FUNCTION_BLOCK FB_Manipulatormodul
VAR_INPUT
	bEnable : BOOL;
	bExecute : BOOL;
	
	pXhome : REAL;
	pYhome : REAL;
	pZhome : REAL;
	
	pXconv : REAL;
	pYconv : REAL;
	pZconv : REAL;
	
	pXscale : REAL;
	pYscale : REAL;
	pZscale : REAL;
	
	pXheat : REAL;
	pYheat : REAL;
	pZheat : REAL;
	
	pX1stor : REAL;
	pX2stor : REAL;
	pX3stor : REAL;
	pX4stor : REAL;
	pYstor : REAL;
	pZstor : REAL;
	
	estateE : eBetriebszustand;
	
	bxEndschalter: BOOL;
	byEndschalter: BOOL;
	bzEndschalter: BOOL;
	bGEndschalter: BOOL;
	
END_VAR
VAR_OUTPUT
	estate : eBetriebszustand;
END_VAR
VAR
	fbRobotsteuerung : FB_Robotsteuerung;
	fbTON : TON;
	nstate : INT := 0;
	
	targX   : REAL;
  	targY   : REAL;
 	targZ   : REAL;
  	goRobot : BOOL;
END_VAR
VAR_IN_OUT
    // Achsen-Referenzen 
    ax_ManX    : AXIS_REF;   
    ax_ManY    : AXIS_REF;   
    ax_ManZ    : AXIS_REF;  
	ax_ManG    : AXIS_REF;   
END_VAR

fbRobotsteuerung(
	bEnable:= , 
	bExecute:= goRobot, 
	bxposition:= targX, 
	byposition:= targY, 
	bzposition:= targZ, 
	bxEndschalter:= bxEndschalter, 
	byEndschalter:= byEndschalter, 
	bzEndschalter:= bzEndschalter, 
	bGEndschalter:= bGEndschalter, 
	estate=> , 
	movedone=> , 
	ax_ManX:= ax_ManX, 
	ax_ManY:= ax_ManY, 
	ax_ManZ:= ax_ManZ, 
	ax_ManG:= ax_ManG);
	
	fbTON(IN:= , PT:=T#10S , Q=> , ET=> );
CASE nstate OF 
	0: //off
	estate := eBetriebszustand.off;
	fbRobotsteuerung.bEnable := FALSE;
	
	IF bEnable THEN
		nstate := 10;
	END_IF
	
	10: //Init
	estate := eBetriebszustand.init;
	fbRobotsteuerung.bEnable := TRUE;
	
	IF fbRobotsteuerung.estate = eBetriebszustand.ready THEN
		nstate := 20;
	END_IF
	
	20: //Ready
	estate := eBetriebszustand.ready;
	fbRobotsteuerung.bEnable := TRUE;
	
	IF bExecute THEN
		nState := 30; 
	END_IF
	
	30: //Move to Conveyer
	estate := eBetriebszustand.production;
	targX   := pXconv;
  	targY   := pYconv;
 	targZ   := pZconv;
  	goRobot := TRUE;
	
	IF fbRobotsteuerung.estate = eBetriebszustand.done AND
		estateE = eBetriebszustand.done THEN
		goRobot := FALSE;
		nstate := 40;
	END_IF
	
	40: //Lift Z Achse
	estate := eBetriebszustand.production;
	targX   := pXconv;
  	targY   := pYconv;
 	targZ   := pZhome;
  	goRobot := TRUE;


	IF fbRobotsteuerung.estate = eBetriebszustand.done THEN
		goRobot := FALSE;
		nstate := 50;
	END_IF
	
	50: //scale
	estate := eBetriebszustand.production;
	targX   := pXscale;
  	targY   := pYscale;
 	targZ   := pZscale;
  	goRobot := TRUE;
	fbTON.IN := TRUE;

	IF fbRobotsteuerung.estate = eBetriebszustand.done AND
		fbTON.Q = TRUE THEN
		fbTON.IN := FALSE;
		goRobot := FALSE;
		nstate := 60;
	END_IF
	
	60: //Lift Z Achse
	estate := eBetriebszustand.production;
	targX   := pXscale;
  	targY   := pYscale;
 	targZ   := pZhome;
  	goRobot := TRUE;

	IF fbRobotsteuerung.estate = eBetriebszustand.done THEN
		goRobot := FALSE;
		nstate := 70;
	END_IF
	
	70: //heat
	estate := eBetriebszustand.production;
	targX   := pXheat;
  	targY   := pYheat;
 	targZ   := pZheat;
  	goRobot := TRUE;
	fbTON.IN := TRUE;
	
	IF fbRobotsteuerung.estate = eBetriebszustand.done AND
		fbTON.Q = TRUE THEN
		fbTON.IN := FALSE;
		goRobot := FALSE;
		nstate := 80;
	END_IF

	80: //Lift Z Achse
	estate := eBetriebszustand.production;
	targX   := pXheat;
  	targY   := pYheat;
 	targZ   := pZhome;
  	goRobot := TRUE;

	IF fbRobotsteuerung.estate = eBetriebszustand.done THEN
		goRobot := FALSE;
		nstate := 90;
	END_IF
	
	90: //storage
	estate := eBetriebszustand.production;
	targX   := pX1stor;
  	targY   := pYstor;
 	targZ   := pZstor;
  	goRobot := TRUE;
	fbTON.IN := TRUE;

	IF fbRobotsteuerung.estate = eBetriebszustand.done AND
		fbTON.Q = TRUE THEN
		fbTON.IN := FALSE;
		goRobot := FALSE;
		nstate := 100;
	END_IF
	
	100: //Lift Z Achse
	estate := eBetriebszustand.production;
	targX   := pX1stor;
  	targY   := pYstor;
 	targZ   := pZhome;
  	goRobot := TRUE;

	IF fbRobotsteuerung.estate = eBetriebszustand.done THEN
		goRobot := FALSE;
		nstate := 110;
	END_IF
	
	110: //Home
	estate := eBetriebszustand.production;
	targX   := pXhome;
  	targY   := pYhome;
 	targZ   := pZhome;
  	goRobot := TRUE;

	IF fbRobotsteuerung.estate = eBetriebszustand.done THEN
		goRobot := FALSE;
		nstate := 120;
	END_IF
	
	120: // Done
	estate:= eBetriebszustand.done;
	fbRobotsteuerung.bExecute := FALSE;
	
	
END_CASE

END_FUNCTION_BLOCK

(* stored: Version 1.1.0.1, ProductVersion 3.1.4024.15
   POU FB_Manipulatormodul: Id {2c2befd5-8aae-4d41-91d7-a7d4b4d4e8de}, SpecialFunc None *)
